Universal Robots PolyScope program: 0603.urp

Program 0603 (installation=default directory=/home/ur/ursim-current/programs/새로운 폴더 createdIn=5.12.7.1102192 lastSavedIn=5.12.7.1102192 robotSerialNumber=20195599999)
Calibrated DH parameters: a=[0, -0.425, -0.3922, 0, 0, 0]; d=[0.1625, 0, 0, 0.1333, 0.0997, 0.0996]; alpha=[1.570796, 0, 0, 1.570796, -1.570796, 0]; deltaTheta=[0, 0, 0, 0, 0, 0]
Robot Program (runOnlyOnce=false)
  Folder Init
    Call Socket_Open
    Call Init_Variables
    MoveJ speed 60 deg/s, acceleration 80 deg/s^2 (useActiveTCP=true) feature=Base
      Waypoint Home: 
  Folder Main Sequence
    Folder Task1:OpenPrinter
      Call Enter_Next_Task
      Loop While (checkContinuously=false) expression=retry_count <= max_retry and task_done == 0
        MoveJ speed 60 deg/s, acceleration 80 deg/s^2 (useActiveTCP=true) feature=Base
          Waypoint AccessToPrinter: 
          Waypoint OpenPrinter: 
          Waypoint RetreatFromPrin: 
        Call Check_Door_Open
        Switch expression=fail_flag
          Case (caseValue=0)
            Script: task_done = 1
          Case (caseValue=1)
            Script: retry_count = retry_count + 1
      If task_done == 0
        Call Error_Stop
    Folder Task2:PickA4FromTray
      Call Enter_Next_Task
      MoveJ speed 60 deg/s, acceleration 80 deg/s^2 (useActiveTCP=true) feature=Base
        Waypoint AccessToTray: 
      Call Gripper_Open
      Call Wait_Motor_Idle
      Call DC_Run
      Call Wait_Motor_Idle
      Call Gripper_Close
      Call Wait_Motor_Idle
      MoveJ speed 60 deg/s, acceleration 80 deg/s^2 (useActiveTCP=true) feature=Base
        Waypoint RetreatFromTray: 
      If fail_flag == 1
        Call Error_Stop
    Folder Task3:PlaceA4OnScanner
      Call Enter_Next_Task
      MoveJ speed 60 deg/s, acceleration 80 deg/s^2 (useActiveTCP=true) feature=Base
        Waypoint AccessToScanne: 
      Call Gripper_Open
      Call Wait_Motor_Idle
      MoveJ speed 60 deg/s, acceleration 80 deg/s^2 (useActiveTCP=true) feature=Base
        Waypoint RetreatFromScan: 
      Call Check_Paper_Detected
      If fail_flag == 1
        Call Error_Stop
    Folder Task4:ClosePrinter
      Call Enter_Next_Task
      Loop While (checkContinuously=false) expression=retry_count <= max_retry and task_done == 0
        MoveJ speed 60 deg/s, acceleration 80 deg/s^2 (useActiveTCP=true) feature=Base
          Waypoint AccessToPrinter: 
          Waypoint ClosePrinterr: 
          Waypoint RetreatFromPrin: 
        Call Check_Door_Closed
        Switch expression=fail_flag
          Case (caseValue=0)
            Script: task_done = 1
          Case (caseValue=1)
            Script: retry_count = retry_count + 1
      If task_done == 0
        Call Error_Stop
    Folder Task5:OpenPrinter
      Call Enter_Next_Task
      Loop While (checkContinuously=false) expression=retry_count <= max_retry and task_done == 0
        MoveJ speed 60 deg/s, acceleration 80 deg/s^2 (useActiveTCP=true) feature=Base
          Waypoint AccessToPrinter: 
          Waypoint OpenPrinterr: 
          Waypoint RetreatFromPrin: 
        Call Check_Door_Open
        Switch expression=fail_flag
          Case (caseValue=0)
            Script: task_done = 1
          Case (caseValue=1)
            Script: retry_count = retry_count + 1
      If task_done == 0
        Call Error_Stop
    Folder Task6:PickA4FromScanner
      Call Enter_Next_Task
      Call Gripper_Open
      Call Wait_Motor_Idle
      MoveJ speed 60 deg/s, acceleration 80 deg/s^2 (useActiveTCP=true) feature=Base
        Waypoint AccessToScanner: 
      Call Gripper_Close
      Call Wait_Motor_Idle
      MoveJ speed 60 deg/s, acceleration 80 deg/s^2 (useActiveTCP=true) feature=Base
        Waypoint RetreatFromSca: 
      If fail_flag == 1
        Call Error_Stop
    Folder Task7:PlaceA4InBasket
      Call Enter_Next_Task
      MoveJ speed 60 deg/s, acceleration 80 deg/s^2 (useActiveTCP=true) feature=Base
        Waypoint AccessToBasket: 
      Call Gripper_Open
      Call Wait_Motor_Idle
      MoveJ speed 60 deg/s, acceleration 80 deg/s^2 (useActiveTCP=true) feature=Base
        Waypoint RetreatFromBask: 
      If fail_flag == 1
        Call Error_Stop
    Folder Task8:ClosePrinter
      Call Enter_Next_Task
      Loop While (checkContinuously=false) expression=retry_count <= max_retry and task_done == 0
        MoveJ speed 60 deg/s, acceleration 80 deg/s^2 (useActiveTCP=true) feature=Base
          Waypoint AccessToPrinter: 
          Waypoint ClosePrinter: 
          Waypoint RetreatFromPrin: 
        Call Check_Door_Closed
        Switch expression=fail_flag
          Case (caseValue=0)
            Script: task_done = 1
          Case (caseValue=1)
            Script: retry_count = retry_count + 1
      If task_done == 0
        Call Error_Stop
SubProgram -> Init_Variables
SubProgram -> Socket_Open
SubProgram -> DC_Run
SubProgram -> Gripper_Close
SubProgram -> Gripper_Open
SubProgram -> Wait_Motor_Idle
SubProgram -> Check_Door_Closed
SubProgram -> Check_Door_Open
SubProgram -> Check_Paper_Detected
SubProgram -> Error_Stop
SubProgram -> Enter_Next_Task
SubProgram Socket_Open (keepSynchronizedWithDisk=false)
  Placeholder
SubProgram Init_Variables (keepSynchronizedWithDisk=false)
  Placeholder
SubProgram Enter_Next_Task (keepSynchronizedWithDisk=false)
  Placeholder
SubProgram Check_Door_Open (keepSynchronizedWithDisk=false)
  Placeholder
SubProgram Error_Stop (keepSynchronizedWithDisk=false)
  Placeholder
SubProgram Gripper_Open (keepSynchronizedWithDisk=false)
  Placeholder
SubProgram Wait_Motor_Idle (keepSynchronizedWithDisk=false)
  Placeholder
SubProgram DC_Run (keepSynchronizedWithDisk=false)
  Placeholder
SubProgram Gripper_Close (keepSynchronizedWithDisk=false)
  Placeholder
SubProgram Check_Paper_Detected (keepSynchronizedWithDisk=false)
  Placeholder
SubProgram Check_Door_Closed (keepSynchronizedWithDisk=false)
  Placeholder
